(* CODESYS project Acionamento da esteira transportadora_RECOVERED_2019-12-09T20-01-45.project

Project tree, tasks and I/O mapping:
  Device : CODESYS Control Win V3, 3S - Smart Software Solutions GmbH, order no. 305021, version 3.5.11.30
    application Application
      libraries: Standard, * (System)
      task MainTask (cyclic, interval t#20ms, priority 1) calls PLC_PRG
      program PLC_PRG [LD]
      Symbols
*)

// Device/Application/PLC_PRG
PROGRAM PLC_PRG
VAR 
	Start:BOOL;
	Stop:BOOL;
	Emergencia:BOOL;
	Sensor:BOOL; 
	Start_Light:BOOL;
	Stop_Light:BOOL;
	Esteira:BOOL;
	
END_VAR

// NETWORK 1

END_PROGRAM
